{attribute addProperty BoxType "EPP6002-0002-0016"}
{attribute addProperty Id "CtrlAT %Q*WORD1621Data_OutAT %Q*ARRAY[0 ..21] OF USINT176220"}
{attribute addProperty CRC "3891160833"}
{attribute addProperty SizeInBites "192"}
{attribute addProperty SizeInBytes "24"}
TYPE COM_RxPDO_Map_Outputs_Channel_CEA6CFDD :
STRUCT
	{attribute addProperty Name "Ctrl"}
	Ctrl AT %Q* : WORD;
	{attribute addProperty Name "Data_Out"}
	Data_Out AT %Q* : ARRAY[0 ..21] OF USINT;
END_STRUCT
END_TYPE

(* stored: Version 1.2.0.0, ProductVersion 3.1.4024.9
   DUT COM_RxPDO_Map_Outputs_Channel_CEA6CFDD: Id {e7c07ecf-9896-4849-91b2-8858ee387c50} *)
